// Mitsubishi GX Works2 project: PART_REPEAT_SEQUENCE   PLC: Q03UDV

PROGRAM MAIN
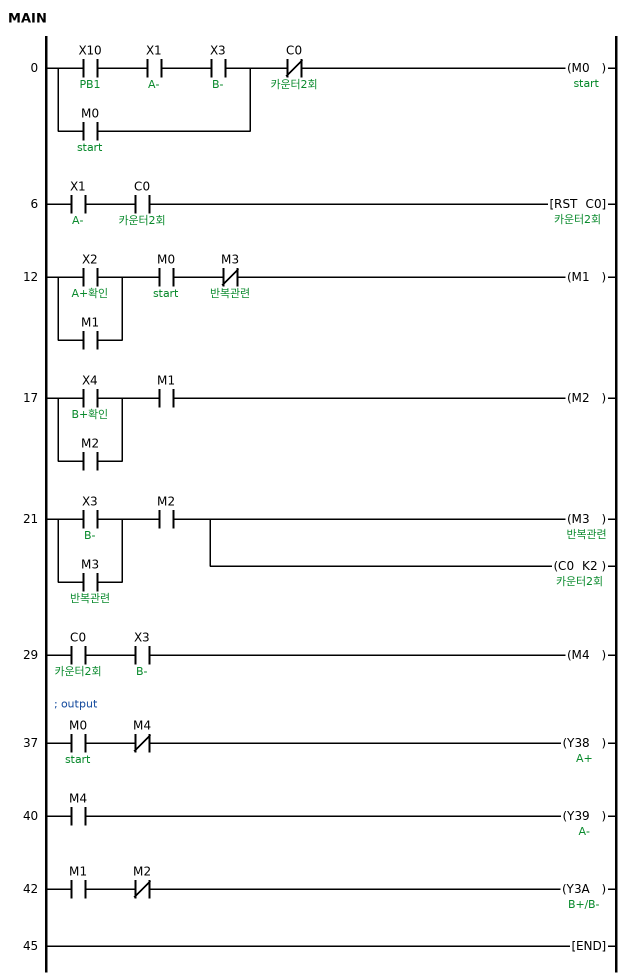
0     LD      X10  ; PB1
      AND     X1  ; A-
      AND     X3  ; B-
      OR      M0  ; start
      ANI     C0  ; 카운터2회
      OUT     M0  ; start
6     LD      X1  ; A-
      AND     C0  ; 카운터2회
      RST     C0  ; 카운터2회
12    LD      X2  ; A+확인
      OR      M1
      AND     M0  ; start
      ANI     M3  ; 반복관련
      OUT     M1
17    LD      X4  ; B+확인
      OR      M2
      AND     M1
      OUT     M2
21    LD      X3  ; B-
      OR      M3  ; 반복관련
      AND     M2
      OUT     M3  ; 반복관련
      OUT     C0 K2  ; 카운터2회
29    LD      C0  ; 카운터2회
      AND     X3  ; B-
      OUT     M4
; output
37    LD      M0  ; start
      ANI     M4
      OUT     Y38  ; A+
40    LD      M4
      OUT     Y39  ; A-
42    LD      M1
      ANI     M2
      OUT     Y3A  ; B+/B-
45    END
END_PROGRAM
